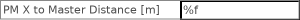
VISUALIZATION _VISU_Pm_Base_Settings  // 300x20
VAR_IN_OUT
	mInst : FB_PrintModule_Base;
END_VAR
    Rectangle (0,0 180x20), "PM X to Master Distance [m]"
    Rectangle (180,0 120x20), "%f", text variable: mInst._fPmDistToMasterRefPos
        OnMouseClick: write the text variable via Default
END_VISUALIZATION

(* stored: Version 1.1.0.1, ProductVersion 3.1.4024.11
   Visu _VISU_Pm_Base_Settings: Id {a1517ad3-9552-4cc0-be69-281725d19d3a} *)
